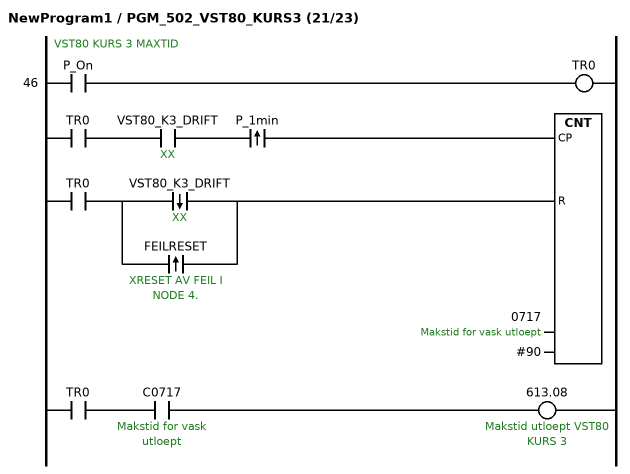
; [picture p552: NewProgram1 / PGM_502_VST80_KURS3, rungs 46-46]
; rung 46: VST80 KURS 3 MAXTID
LD P_On
OUT TR0
AND VST80_K3_DRIFT  ; XX
@AND P_1min
LD TR0
%LD VST80_K3_DRIFT  ; XX
@OR FEILRESET  ; XRESET AV FEIL I NODE 4.
ANDLD
CNT 0717 #90  ; Makstid for vask utloept
LD TR0
AND C0717  ; Makstid for vask utloept
OUT 613.08  ; Makstid utloept VST80 KURS 3

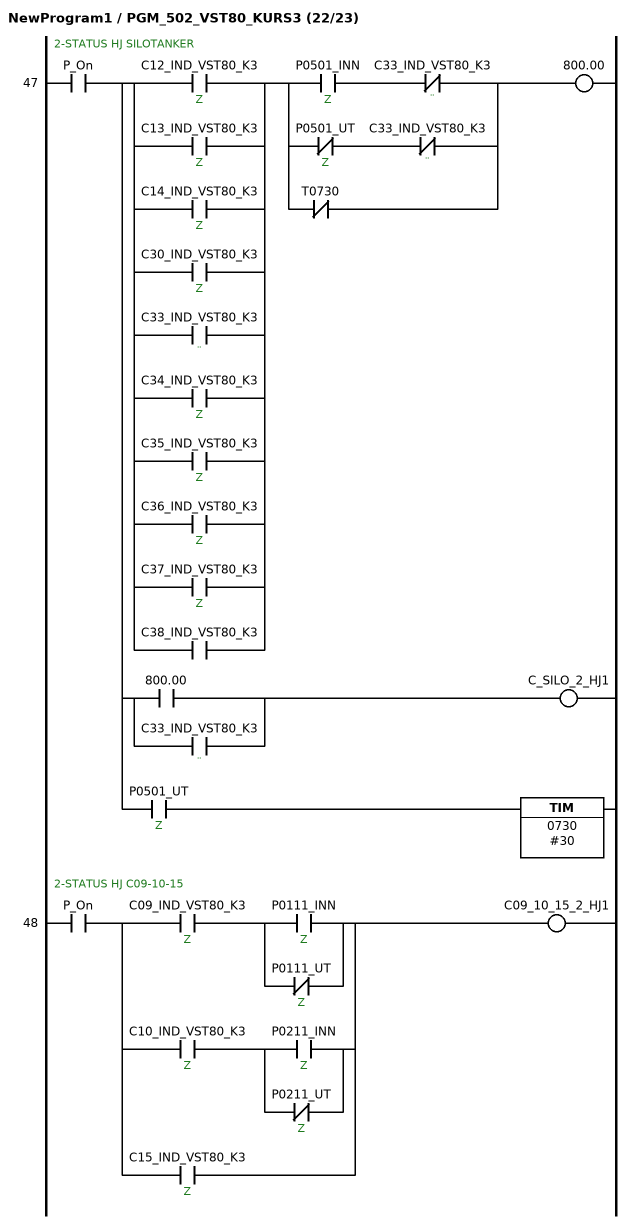
; rung 47: 2-STATUS HJ SILOTANKER
LD P_On
OUT TR0
LD C12_IND_VST80_K3  ; Z
OR C13_IND_VST80_K3  ; Z
OR C14_IND_VST80_K3  ; Z
OR C30_IND_VST80_K3  ; Z
OR C33_IND_VST80_K3  ; ¨
OR C34_IND_VST80_K3  ; Z
OR C35_IND_VST80_K3  ; Z
OR C36_IND_VST80_K3  ; Z
OR C37_IND_VST80_K3  ; Z
OR C38_IND_VST80_K3
ANDLD
LD P0501_INN  ; Z
ANDNOT C33_IND_VST80_K3  ; ¨
LDNOT P0501_UT  ; Z
ANDNOT C33_IND_VST80_K3  ; ¨
ORLD
ORNOT T0730
ANDLD
OUT 800.00
LD TR0
LD 800.00
OR C33_IND_VST80_K3  ; ¨
ANDLD
OUT C_SILO_2_HJ1
LD TR0
AND P0501_UT  ; Z
TIM 0730 #30
; rung 48: 2-STATUS HJ C09-10-15
LD P_On
LD C09_IND_VST80_K3  ; Z
LD P0111_INN  ; Z
ORNOT P0111_UT  ; Z
ANDLD
LD C10_IND_VST80_K3  ; Z
LD P0211_INN  ; Z
ORNOT P0211_UT  ; Z
ANDLD
ORLD
OR C15_IND_VST80_K3  ; Z
ANDLD
OUT C09_10_15_2_HJ1

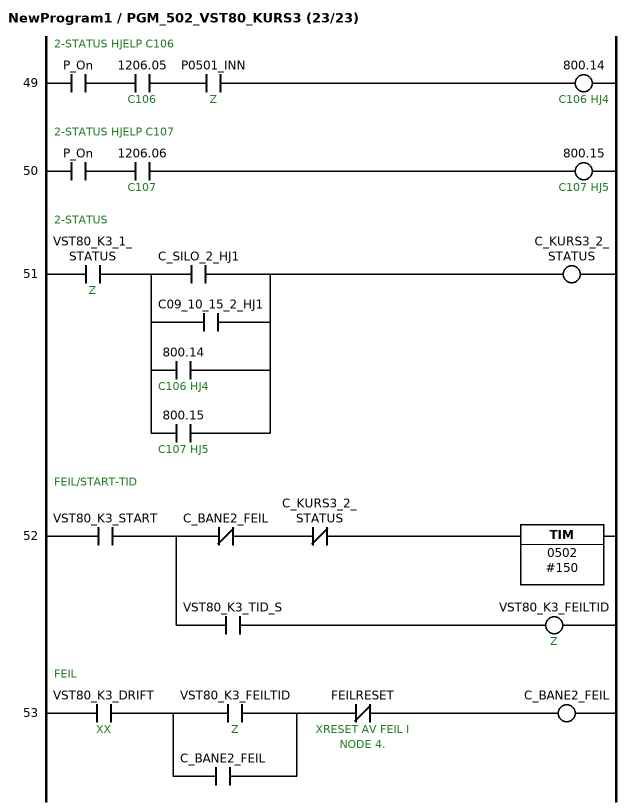
; rung 49: 2-STATUS HJELP C106
LD P_On
AND 1206.05  ; C106
AND P0501_INN  ; Z
OUT 800.14  ; C106 HJ4
; rung 50: 2-STATUS HJELP C107
LD P_On
AND 1206.06  ; C107
OUT 800.15  ; C107 HJ5
; rung 51: 2-STATUS
LD VST80_K3_1_STATUS  ; Z
LD C_SILO_2_HJ1
OR C09_10_15_2_HJ1
OR 800.14  ; C106 HJ4
OR 800.15  ; C107 HJ5
ANDLD
OUT C_KURS3_2_STATUS
; rung 52: FEIL/START-TID
LD VST80_K3_START
OUT TR0
ANDNOT C_BANE2_FEIL
ANDNOT C_KURS3_2_STATUS
TIM 0502 #150
LD TR0
AND VST80_K3_TID_S
OUT VST80_K3_FEILTID  ; Z
; rung 53: FEIL
LD VST80_K3_DRIFT  ; XX
LD VST80_K3_FEILTID  ; Z
OR C_BANE2_FEIL
ANDLD
ANDNOT FEILRESET  ; XRESET AV FEIL I NODE 4.
OUT C_BANE2_FEIL
; rung 54: Ingen_kommentar_funnet

### Section PGM503_C23

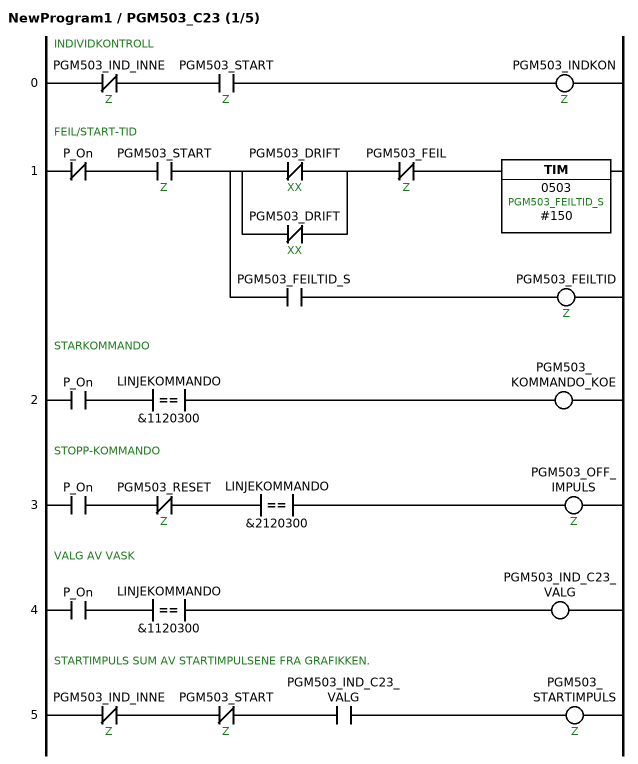
; rung 0: INDIVIDKONTROLL
LDNOT PGM503_IND_INNE  ; Z
AND PGM503_START  ; Z
OUT PGM503_INDKON  ; Z
; rung 1: FEIL/START-TID
LDNOT P_On
AND PGM503_START  ; Z
OUT TR0
LDNOT PGM503_DRIFT  ; XX
ORNOT PGM503_DRIFT  ; XX
ANDLD
ANDNOT PGM503_FEIL  ; Z
TIM 0503 #150  ; PGM503_FEILTID_S
LD TR0
AND PGM503_FEILTID_S
OUT PGM503_FEILTID  ; Z
; rung 2: STARKOMMANDO
LD P_On
AND=L(301) LINJEKOMMANDO &1120300
OUT PGM503_KOMMANDO_KOE
; rung 3: STOPP-KOMMANDO
LD P_On
ANDNOT PGM503_RESET  ; Z
AND=L(301) LINJEKOMMANDO &2120300
OUT PGM503_OFF_IMPULS  ; Z
; rung 4: VALG AV VASK
LD P_On
AND=L(301) LINJEKOMMANDO &1120300
OUT PGM503_IND_C23_VALG
; rung 5: STARTIMPULS SUM AV STARTIMPULSENE FRA GRAFIKKEN.
LDNOT PGM503_IND_INNE  ; Z
ANDNOT PGM503_START  ; Z
AND PGM503_IND_C23_VALG
OUT PGM503_STARTIMPULS  ; Z

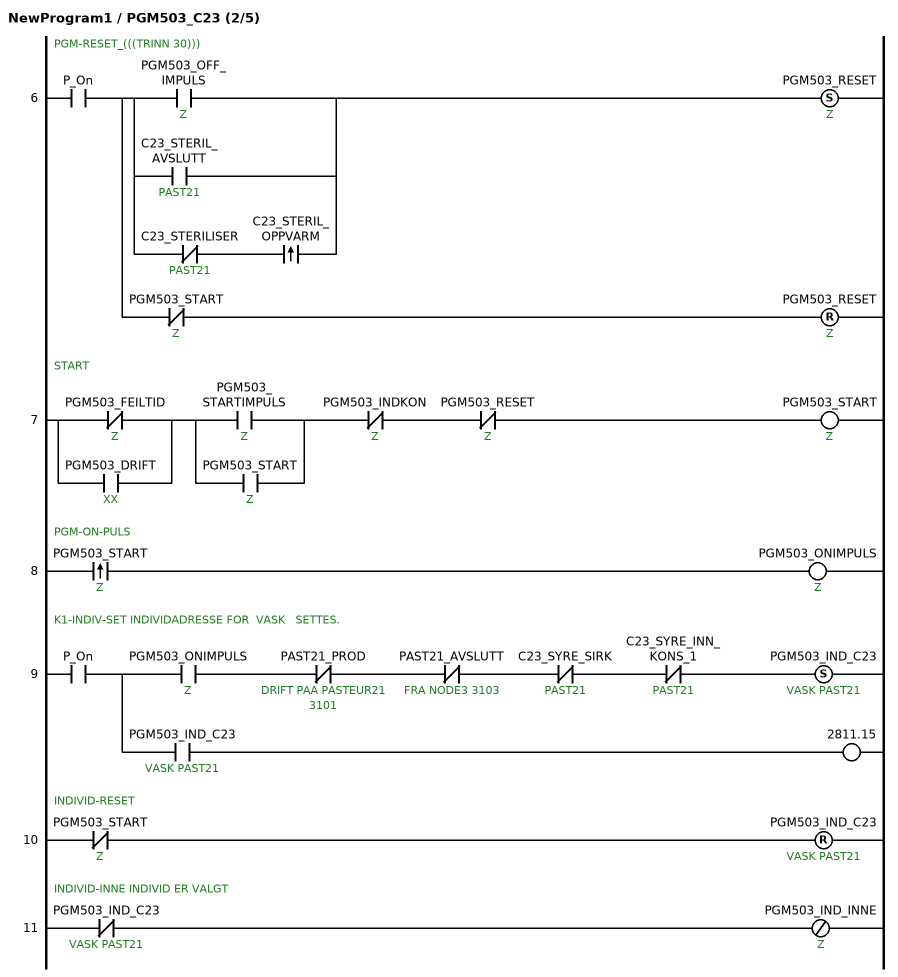
; rung 6: PGM-RESET_(((TRINN 30)))
LD P_On
OUT TR0
LD PGM503_OFF_IMPULS  ; Z
OR C23_STERIL_AVSLUTT  ; PAST21
LDNOT C23_STERILISER  ; PAST21
@AND C23_STERIL_OPPVARM
ORLD
ANDLD
SET PGM503_RESET  ; Z
LD TR0
ANDNOT PGM503_START  ; Z
RSET PGM503_RESET  ; Z
; rung 7: START
LDNOT PGM503_FEILTID  ; Z
OR PGM503_DRIFT  ; XX
LD PGM503_STARTIMPULS  ; Z
OR PGM503_START  ; Z
ANDLD
ANDNOT PGM503_INDKON  ; Z
ANDNOT PGM503_RESET  ; Z
OUT PGM503_START  ; Z
; rung 8: PGM-ON-PULS
@LD PGM503_START  ; Z
OUT PGM503_ONIMPULS  ; Z
; rung 9: K1-INDIV-SET INDIVIDADRESSE FOR  VASK   SETTES.
LD P_On
OUT TR0
AND PGM503_ONIMPULS  ; Z
ANDNOT PAST21_PROD  ; DRIFT PAA PASTEUR21 3101
ANDNOT PAST21_AVSLUTT  ; FRA NODE3 3103
ANDNOT C23_SYRE_SIRK  ; PAST21
ANDNOT C23_SYRE_INN_KONS_1  ; PAST21
SET PGM503_IND_C23  ; VASK PAST21
LD TR0
AND PGM503_IND_C23  ; VASK PAST21
OUT 2811.15
; rung 10: INDIVID-RESET
LDNOT PGM503_START  ; Z
RSET PGM503_IND_C23  ; VASK PAST21
; rung 11: INDIVID-INNE INDIVID ER VALGT
LDNOT PGM503_IND_C23  ; VASK PAST21
OUTNOT PGM503_IND_INNE  ; Z

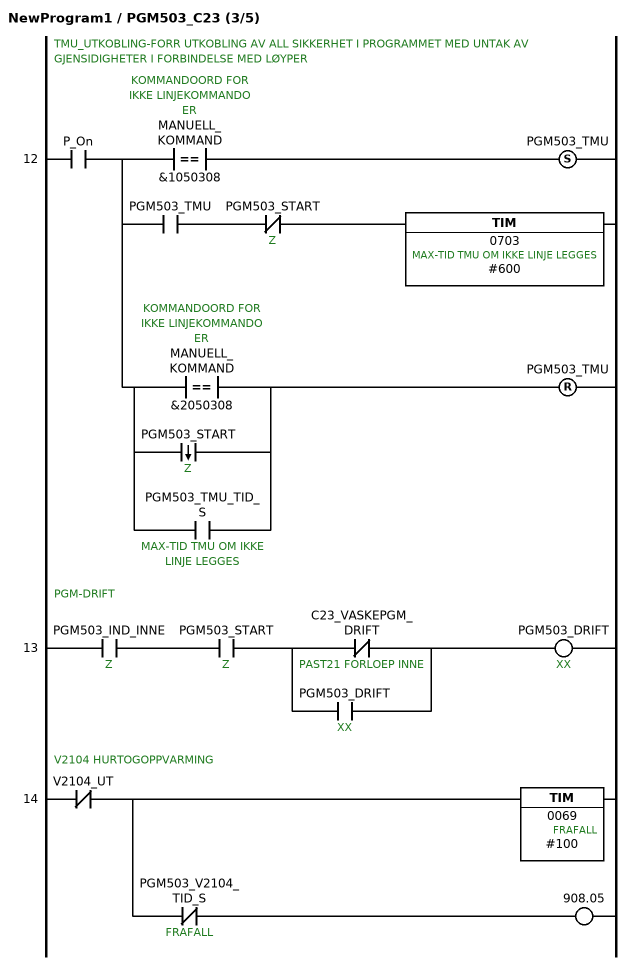
; rung 12: TMU_UTKOBLING-FORR UTKOBLING AV ALL SIKKERHET I PROGRAMMET MED UNTAK AV GJENSIDIGHETER I FORBINDELSE MED LØYPER
LD P_On
OUT TR0
AND=L(301) MANUELL_KOMMAND &1050308  ; KOMMANDOORD FOR IKKE LINJEKOMMANDOER
SET PGM503_TMU
LD TR0
AND PGM503_TMU
ANDNOT PGM503_START  ; Z
TIM 0703 #600  ; MAX-TID TMU OM IKKE LINJE LEGGES
LD TR0
LD=L(301) MANUELL_KOMMAND &2050308  ; KOMMANDOORD FOR IKKE LINJEKOMMANDOER
%OR PGM503_START  ; Z
OR PGM503_TMU_TID_S  ; MAX-TID TMU OM IKKE LINJE LEGGES
ANDLD
RSET PGM503_TMU
; rung 13: PGM-DRIFT
LD PGM503_IND_INNE  ; Z
AND PGM503_START  ; Z
LDNOT C23_VASKEPGM_DRIFT  ; PAST21 FORLOEP INNE
OR PGM503_DRIFT  ; XX
ANDLD
OUT PGM503_DRIFT  ; XX
; rung 14: V2104 HURTOGOPPVARMING
LDNOT V2104_UT
TIM 0069 #100  ; FRAFALL
ANDNOT PGM503_V2104_TID_S  ; FRAFALL
OUT 908.05

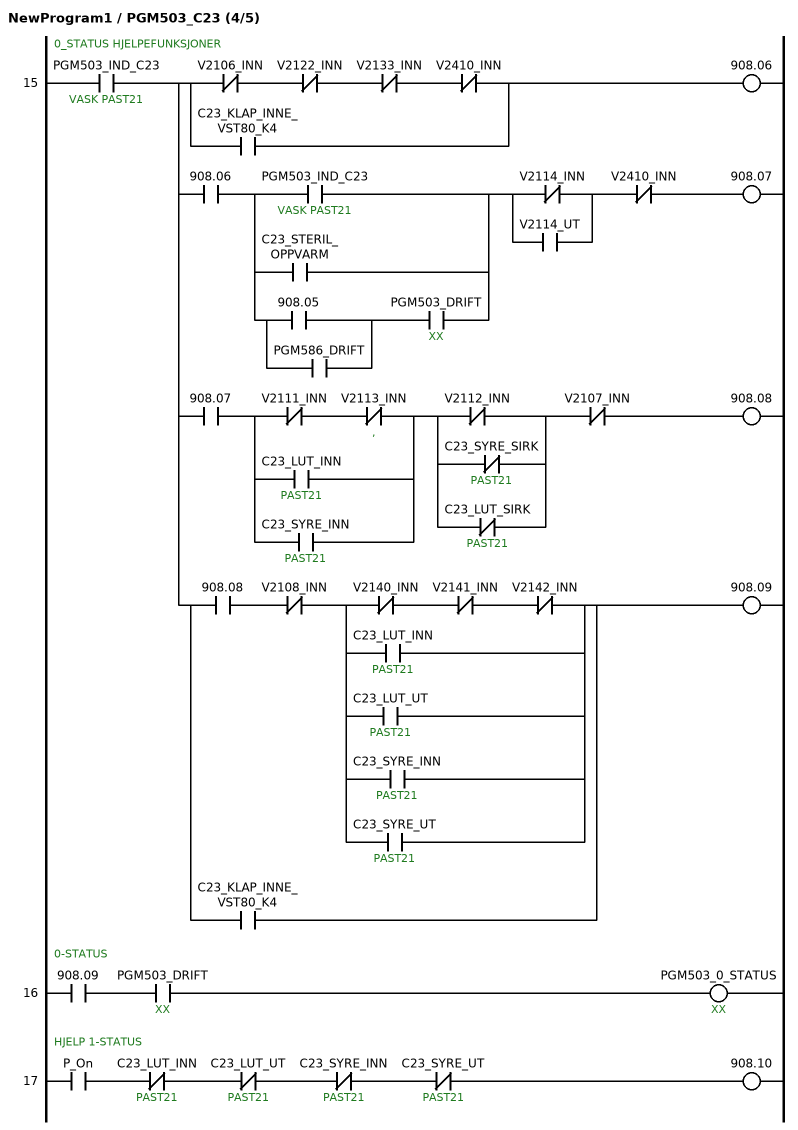
; rung 15: 0_STATUS HJELPEFUNKSJONER
LD PGM503_IND_C23  ; VASK PAST21
OUT TR0
LDNOT V2106_INN
ANDNOT V2122_INN
ANDNOT V2133_INN
ANDNOT V2410_INN
OR C23_KLAP_INNE_VST80_K4
ANDLD
OUT 908.06
LD TR0
AND 908.06
LD PGM503_IND_C23  ; VASK PAST21
OR C23_STERIL_OPPVARM
LD 908.05
OR PGM586_DRIFT
AND PGM503_DRIFT  ; XX
ORLD
ANDLD
LDNOT V2114_INN
OR V2114_UT
ANDLD
ANDNOT V2410_INN
OUT 908.07
LD TR0
AND 908.07
LDNOT V2111_INN
ANDNOT V2113_INN  ; ,
OR C23_LUT_INN  ; PAST21
OR C23_SYRE_INN  ; PAST21
ANDLD
LDNOT V2112_INN
ORNOT C23_SYRE_SIRK  ; PAST21
ORNOT C23_LUT_SIRK  ; PAST21
ANDLD
ANDNOT V2107_INN
OUT 908.08
LD TR0
LD 908.08
ANDNOT V2108_INN
LDNOT V2140_INN
ANDNOT V2141_INN
ANDNOT V2142_INN
OR C23_LUT_INN  ; PAST21
OR C23_LUT_UT  ; PAST21
OR C23_SYRE_INN  ; PAST21
OR C23_SYRE_UT  ; PAST21
ANDLD
OR C23_KLAP_INNE_VST80_K4
ANDLD
OUT 908.09
; rung 16: 0-STATUS
LD 908.09
AND PGM503_DRIFT  ; XX
OUT PGM503_0_STATUS  ; XX
; rung 17: HJELP 1-STATUS
LD P_On
ANDNOT C23_LUT_INN  ; PAST21
ANDNOT C23_LUT_UT  ; PAST21
ANDNOT C23_SYRE_INN  ; PAST21
ANDNOT C23_SYRE_UT  ; PAST21
OUT 908.10

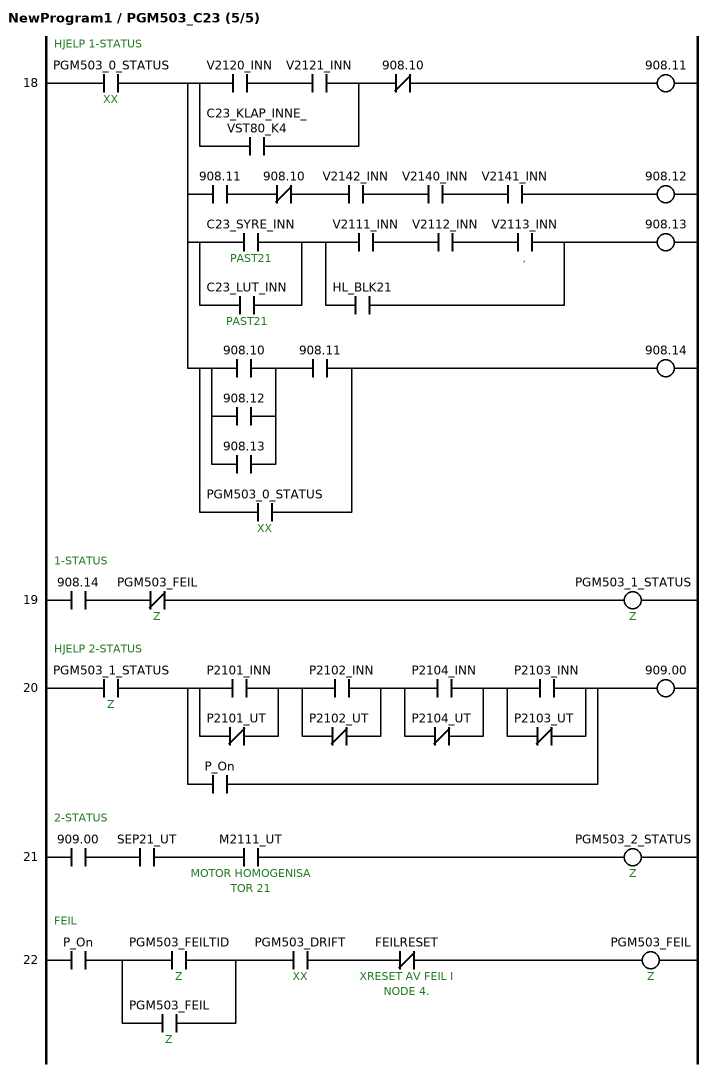
; rung 18: HJELP 1-STATUS
LD PGM503_0_STATUS  ; XX
OUT TR0
LD V2120_INN
AND V2121_INN
OR C23_KLAP_INNE_VST80_K4
ANDLD
ANDNOT 908.10
OUT 908.11
LD TR0
AND 908.11
ANDNOT 908.10
AND V2142_INN
AND V2140_INN
AND V2141_INN
OUT 908.12
LD TR0
LD C23_SYRE_INN  ; PAST21
OR C23_LUT_INN  ; PAST21
ANDLD
LD V2111_INN
AND V2112_INN
AND V2113_INN  ; ,
OR HL_BLK21
ANDLD
OUT 908.13
LD TR0
LD 908.10
OR 908.12
OR 908.13
AND 908.11
OR PGM503_0_STATUS  ; XX
ANDLD
OUT 908.14
; rung 19: 1-STATUS
LD 908.14
ANDNOT PGM503_FEIL  ; Z
OUT PGM503_1_STATUS  ; Z
; rung 20: HJELP 2-STATUS
LD PGM503_1_STATUS  ; Z
LD P2101_INN
ORNOT P2101_UT
LD P2102_INN
ORNOT P2102_UT
ANDLD
LD P2104_INN
ORNOT P2104_UT
ANDLD
LD P2103_INN
ORNOT P2103_UT
ANDLD
OR P_On
ANDLD
OUT 909.00
; rung 21: 2-STATUS
LD 909.00
AND SEP21_UT
AND M2111_UT  ; MOTOR HOMOGENISATOR 21
OUT PGM503_2_STATUS  ; Z
; rung 22: FEIL
LD P_On
LD PGM503_FEILTID  ; Z
OR PGM503_FEIL  ; Z
ANDLD
AND PGM503_DRIFT  ; XX
ANDNOT FEILRESET  ; XRESET AV FEIL I NODE 4.
OUT PGM503_FEIL  ; Z
; rung 23: Ingen_kommentar_funnet

### Section C23_KLAPRING

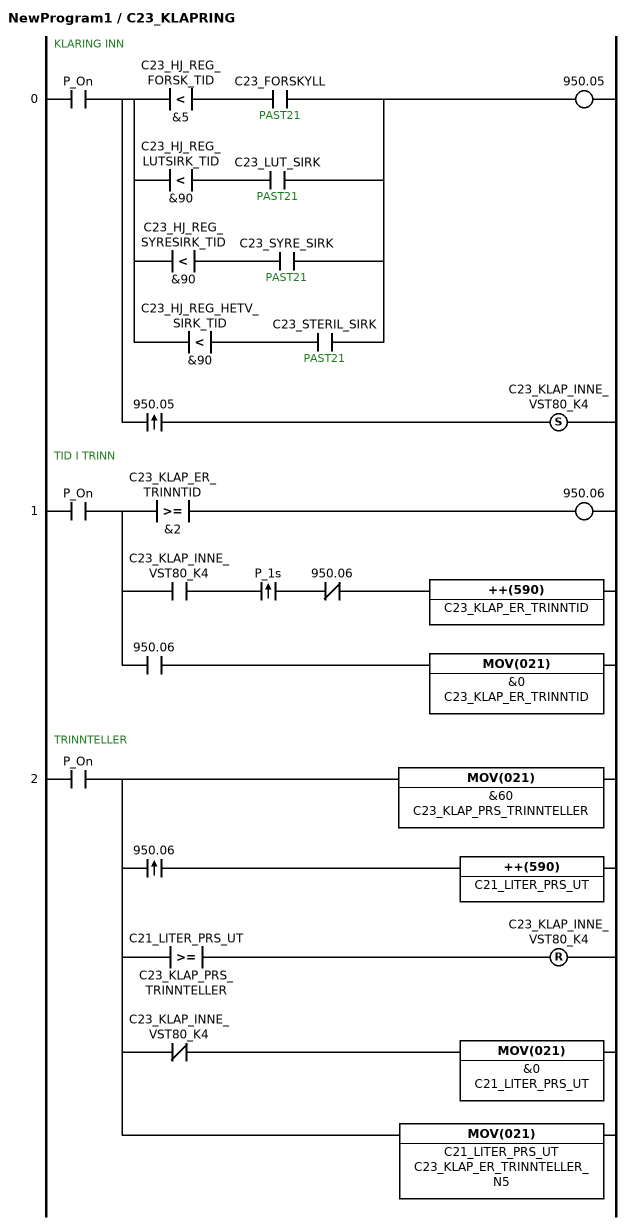
; rung 0: KLARING INN
LD P_On
OUT TR0
LD<(310) C23_HJ_REG_FORSK_TID &5
AND C23_FORSKYLL  ; PAST21
LD<(310) C23_HJ_REG_LUTSIRK_TID &90
AND C23_LUT_SIRK  ; PAST21
ORLD
LD<(310) C23_HJ_REG_SYRESIRK_TID &90
AND C23_SYRE_SIRK  ; PAST21
ORLD
LD<(310) C23_HJ_REG_HETV_SIRK_TID &90
AND C23_STERIL_SIRK  ; PAST21
ORLD
ANDLD
OUT 950.05
LD TR0
@AND 950.05
SET C23_KLAP_INNE_VST80_K4
; rung 1: TID I TRINN
LD P_On
OUT TR0
AND>=(325) C23_KLAP_ER_TRINNTID &2
OUT 950.06
LD TR0
AND C23_KLAP_INNE_VST80_K4
@AND P_1s
ANDNOT 950.06
++(590) C23_KLAP_ER_TRINNTID
LD TR0
AND 950.06
MOV(021) &0 C23_KLAP_ER_TRINNTID
; rung 2: TRINNTELLER
LD P_On
OUT TR0
MOV(021) &60 C23_KLAP_PRS_TRINNTELLER
@AND 950.06
++(590) C21_LITER_PRS_UT
LD TR0
AND>=(325) C21_LITER_PRS_UT C23_KLAP_PRS_TRINNTELLER
RSET C23_KLAP_INNE_VST80_K4
LD TR0
ANDNOT C23_KLAP_INNE_VST80_K4
MOV(021) &0 C21_LITER_PRS_UT
LD TR0
MOV(021) C21_LITER_PRS_UT C23_KLAP_ER_TRINNTELLER_N5
; rung 3: Ingen_kommentar_funnet

### Section PGM504_C24

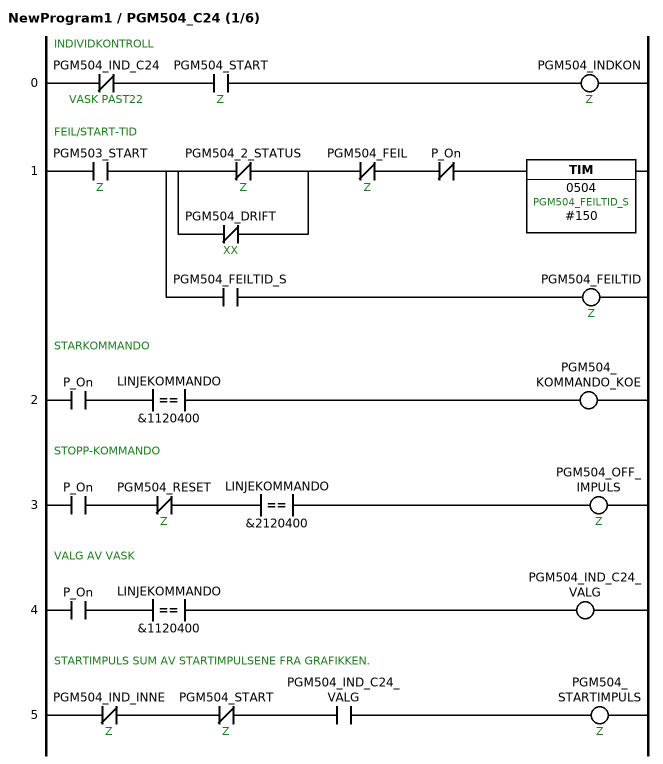
; rung 0: INDIVIDKONTROLL
LDNOT PGM504_IND_C24  ; VASK PAST22
AND PGM504_START  ; Z
OUT PGM504_INDKON  ; Z
; rung 1: FEIL/START-TID
LD PGM503_START  ; Z
OUT TR0
LDNOT PGM504_2_STATUS  ; Z
ORNOT PGM504_DRIFT  ; XX
ANDLD
ANDNOT PGM504_FEIL  ; Z
ANDNOT P_On
TIM 0504 #150  ; PGM504_FEILTID_S
LD TR0
AND PGM504_FEILTID_S
OUT PGM504_FEILTID  ; Z
; rung 2: STARKOMMANDO
LD P_On
AND=L(301) LINJEKOMMANDO &1120400
OUT PGM504_KOMMANDO_KOE
; rung 3: STOPP-KOMMANDO
LD P_On
ANDNOT PGM504_RESET  ; Z
AND=L(301) LINJEKOMMANDO &2120400
OUT PGM504_OFF_IMPULS  ; Z
; rung 4: VALG AV VASK
LD P_On
AND=L(301) LINJEKOMMANDO &1120400
OUT PGM504_IND_C24_VALG
; rung 5: STARTIMPULS SUM AV STARTIMPULSENE FRA GRAFIKKEN.
LDNOT PGM504_IND_INNE  ; Z
ANDNOT PGM504_START  ; Z
AND PGM504_IND_C24_VALG
OUT PGM504_STARTIMPULS  ; Z

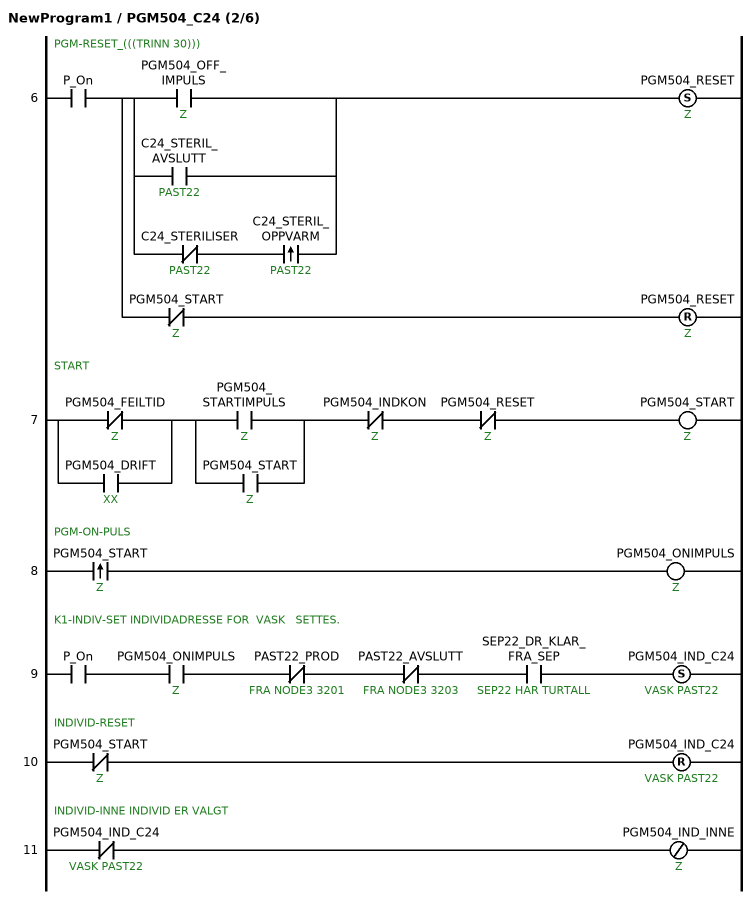
; rung 6: PGM-RESET_(((TRINN 30)))
LD P_On
OUT TR0
LD PGM504_OFF_IMPULS  ; Z
OR C24_STERIL_AVSLUTT  ; PAST22
LDNOT C24_STERILISER  ; PAST22
@AND C24_STERIL_OPPVARM  ; PAST22
ORLD
ANDLD
SET PGM504_RESET  ; Z
LD TR0
ANDNOT PGM504_START  ; Z
RSET PGM504_RESET  ; Z
; rung 7: START
LDNOT PGM504_FEILTID  ; Z
OR PGM504_DRIFT  ; XX
LD PGM504_STARTIMPULS  ; Z
OR PGM504_START  ; Z
ANDLD
ANDNOT PGM504_INDKON  ; Z
ANDNOT PGM504_RESET  ; Z
OUT PGM504_START  ; Z
; rung 8: PGM-ON-PULS
@LD PGM504_START  ; Z
OUT PGM504_ONIMPULS  ; Z
; rung 9: K1-INDIV-SET INDIVIDADRESSE FOR  VASK   SETTES.
LD P_On
AND PGM504_ONIMPULS  ; Z
ANDNOT PAST22_PROD  ; FRA NODE3 3201
ANDNOT PAST22_AVSLUTT  ; FRA NODE3 3203
AND SEP22_DR_KLAR_FRA_SEP  ; SEP22 HAR TURTALL
SET PGM504_IND_C24  ; VASK PAST22
; rung 10: INDIVID-RESET
LDNOT PGM504_START  ; Z
RSET PGM504_IND_C24  ; VASK PAST22
; rung 11: INDIVID-INNE INDIVID ER VALGT
LDNOT PGM504_IND_C24  ; VASK PAST22
OUTNOT PGM504_IND_INNE  ; Z

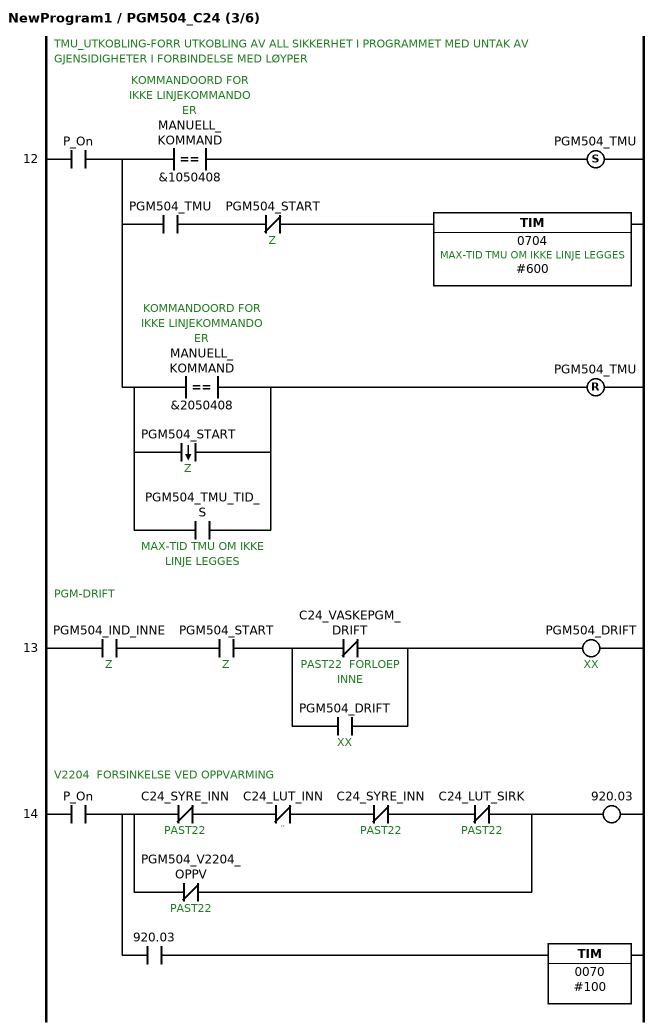
; rung 12: TMU_UTKOBLING-FORR UTKOBLING AV ALL SIKKERHET I PROGRAMMET MED UNTAK AV GJENSIDIGHETER I FORBINDELSE MED LØYPER
LD P_On
OUT TR0
AND=L(301) MANUELL_KOMMAND &1050408  ; KOMMANDOORD FOR IKKE LINJEKOMMANDOER
SET PGM504_TMU
LD TR0
AND PGM504_TMU
ANDNOT PGM504_START  ; Z
TIM 0704 #600  ; MAX-TID TMU OM IKKE LINJE LEGGES
LD TR0
LD=L(301) MANUELL_KOMMAND &2050408  ; KOMMANDOORD FOR IKKE LINJEKOMMANDOER
%OR PGM504_START  ; Z
OR PGM504_TMU_TID_S  ; MAX-TID TMU OM IKKE LINJE LEGGES
ANDLD
RSET PGM504_TMU
; rung 13: PGM-DRIFT
LD PGM504_IND_INNE  ; Z
AND PGM504_START  ; Z
LDNOT C24_VASKEPGM_DRIFT  ; PAST22  FORLOEP INNE
OR PGM504_DRIFT  ; XX
ANDLD
OUT PGM504_DRIFT  ; XX
; rung 14: V2204  FORSINKELSE VED OPPVARMING
LD P_On
OUT TR0
LDNOT C24_SYRE_INN  ; PAST22
ANDNOT C24_LUT_INN  ; ¨
ANDNOT C24_SYRE_INN  ; PAST22
ANDNOT C24_LUT_SIRK  ; PAST22
ORNOT PGM504_V2204_OPPV  ; PAST22
ANDLD
OUT 920.03
LD TR0
AND 920.03
TIM 0070 #100

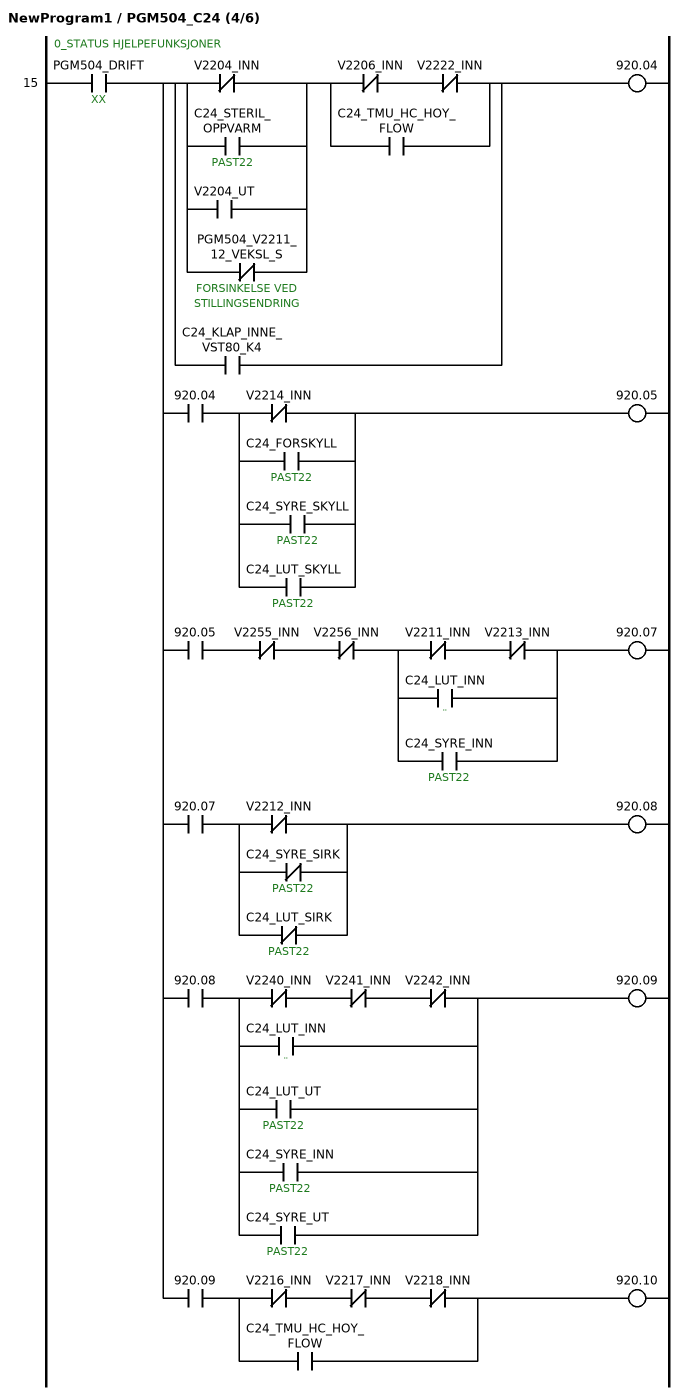
; rung 15: 0_STATUS HJELPEFUNKSJONER
LD PGM504_DRIFT  ; XX
OUT TR0
LDNOT V2204_INN
OR C24_STERIL_OPPVARM  ; PAST22
OR V2204_UT
ORNOT PGM504_V2211_12_VEKSL_S  ; FORSINKELSE VED STILLINGSENDRING
LDNOT V2206_INN
ANDNOT V2222_INN
OR C24_TMU_HC_HOY_FLOW
ANDLD
OR C24_KLAP_INNE_VST80_K4
ANDLD
OUT 920.04
LD TR0
AND 920.04
LDNOT V2214_INN
OR C24_FORSKYLL  ; PAST22
OR C24_SYRE_SKYLL  ; PAST22
OR C24_LUT_SKYLL  ; PAST22
ANDLD
OUT 920.05
LD TR0
AND 920.05
ANDNOT V2255_INN
ANDNOT V2256_INN
LDNOT V2211_INN
ANDNOT V2213_INN
OR C24_LUT_INN  ; ¨
OR C24_SYRE_INN  ; PAST22
ANDLD
OUT 920.07
LD TR0
AND 920.07
LDNOT V2212_INN
ORNOT C24_SYRE_SIRK  ; PAST22
ORNOT C24_LUT_SIRK  ; PAST22
ANDLD
OUT 920.08
LD TR0
AND 920.08
LDNOT V2240_INN
ANDNOT V2241_INN
ANDNOT V2242_INN
OR C24_LUT_INN  ; ¨
OR C24_LUT_UT  ; PAST22
OR C24_SYRE_INN  ; PAST22
OR C24_SYRE_UT  ; PAST22
ANDLD
OUT 920.09
LD TR0
AND 920.09
LDNOT V2216_INN
ANDNOT V2217_INN
ANDNOT V2218_INN
OR C24_TMU_HC_HOY_FLOW
ANDLD
OUT 920.10

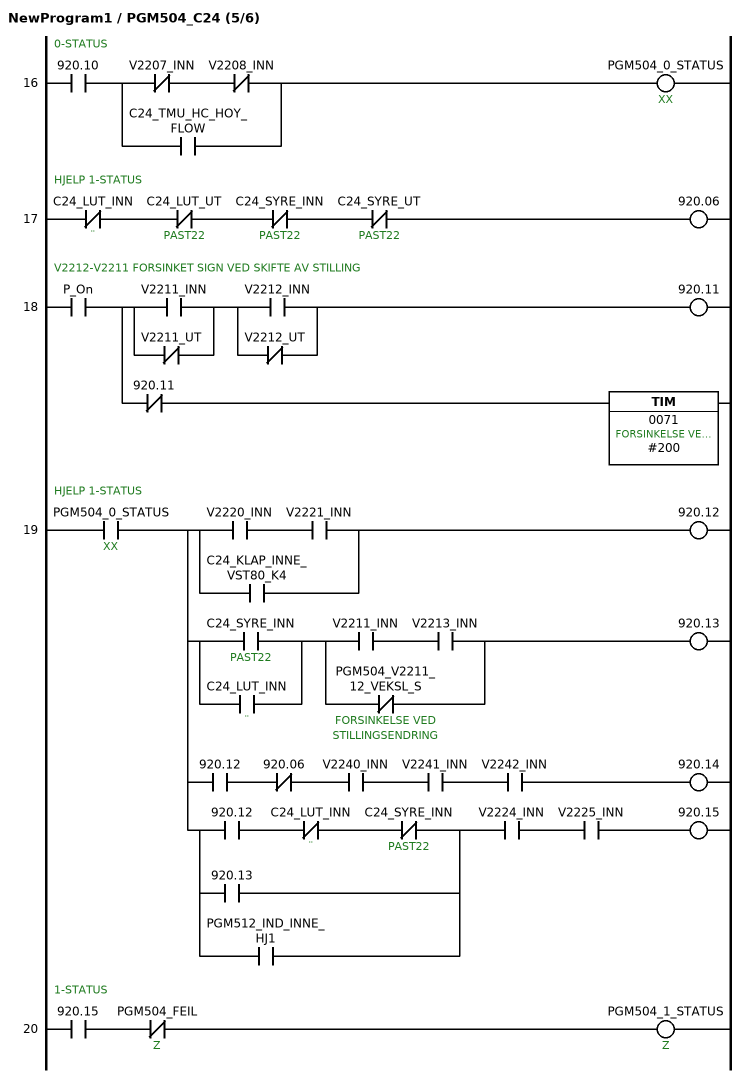
; rung 16: 0-STATUS
LD 920.10
LDNOT V2207_INN
ANDNOT V2208_INN
OR C24_TMU_HC_HOY_FLOW
ANDLD
OUT PGM504_0_STATUS  ; XX
; rung 17: HJELP 1-STATUS
LDNOT C24_LUT_INN  ; ¨
ANDNOT C24_LUT_UT  ; PAST22
ANDNOT C24_SYRE_INN  ; PAST22
ANDNOT C24_SYRE_UT  ; PAST22
OUT 920.06
; rung 18: V2212-V2211 FORSINKET SIGN VED SKIFTE AV STILLING
LD P_On
OUT TR0
LD V2211_INN
ORNOT V2211_UT
ANDLD
LD V2212_INN
ORNOT V2212_UT
ANDLD
OUT 920.11
LD TR0
ANDNOT 920.11
TIM 0071 #200  ; FORSINKELSE VED STILLINGSENDRING
; rung 19: HJELP 1-STATUS
LD PGM504_0_STATUS  ; XX
OUT TR0
LD V2220_INN
AND V2221_INN
OR C24_KLAP_INNE_VST80_K4
ANDLD
OUT 920.12
LD TR0
LD C24_SYRE_INN  ; PAST22
OR C24_LUT_INN  ; ¨
ANDLD
LD V2211_INN
AND V2213_INN
ORNOT PGM504_V2211_12_VEKSL_S  ; FORSINKELSE VED STILLINGSENDRING
ANDLD
OUT 920.13
LD TR0
AND 920.12
ANDNOT 920.06
AND V2240_INN
AND V2241_INN
AND V2242_INN
OUT 920.14
LD TR0
LD 920.12
ANDNOT C24_LUT_INN  ; ¨
ANDNOT C24_SYRE_INN  ; PAST22
OR 920.13
OR PGM512_IND_INNE_HJ1
ANDLD
AND V2224_INN
AND V2225_INN
OUT 920.15
; rung 20: 1-STATUS
LD 920.15
ANDNOT PGM504_FEIL  ; Z
OUT PGM504_1_STATUS  ; Z

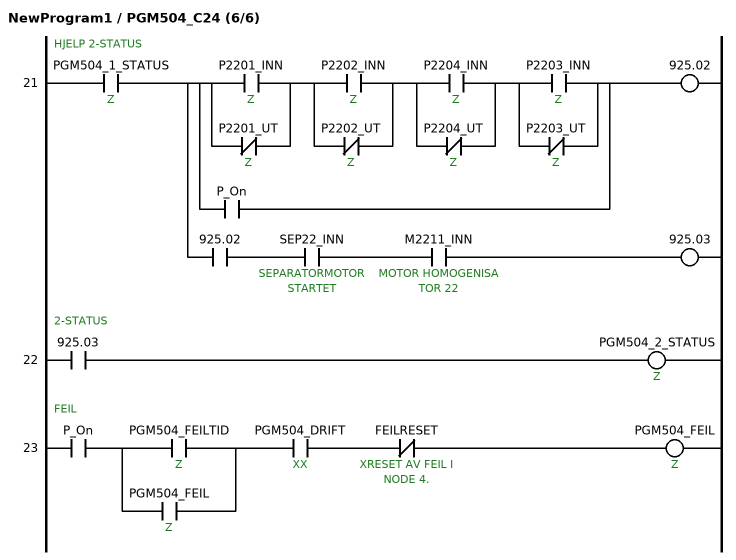
; rung 21: HJELP 2-STATUS
LD PGM504_1_STATUS  ; Z
OUT TR0
LD P2201_INN  ; Z
ORNOT P2201_UT  ; Z
LD P2202_INN  ; Z
ORNOT P2202_UT  ; Z
ANDLD
LD P2204_INN  ; Z
ORNOT P2204_UT  ; Z
ANDLD
LD P2203_INN  ; Z
ORNOT P2203_UT  ; Z
ANDLD
OR P_On
ANDLD
OUT 925.02
LD TR0
AND 925.02
AND SEP22_INN  ; SEPARATORMOTOR STARTET
AND M2211_INN  ; MOTOR HOMOGENISATOR 22
OUT 925.03
; rung 22: 2-STATUS
LD 925.03
OUT PGM504_2_STATUS  ; Z
; rung 23: FEIL
LD P_On
LD PGM504_FEILTID  ; Z
OR PGM504_FEIL  ; Z
ANDLD
AND PGM504_DRIFT  ; XX
ANDNOT FEILRESET  ; XRESET AV FEIL I NODE 4.
OUT PGM504_FEIL  ; Z
; rung 24: Ingen_kommentar_funnet

### Section C24_KLAPRING

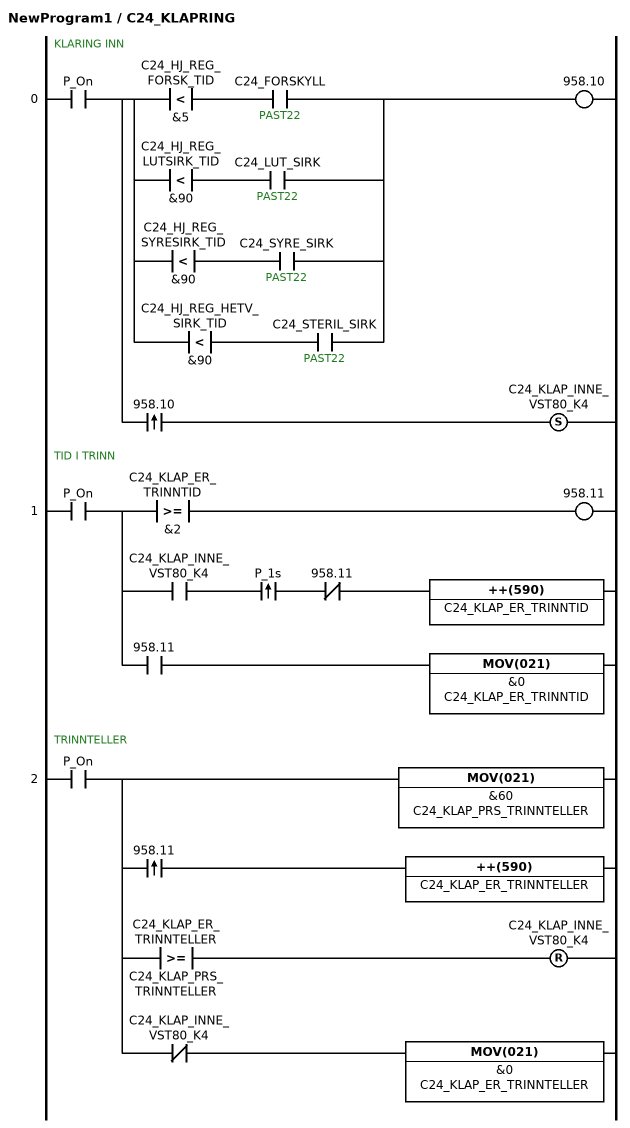
; rung 0: KLARING INN
LD P_On
OUT TR0
LD<(310) C24_HJ_REG_FORSK_TID &5
AND C24_FORSKYLL  ; PAST22
LD<(310) C24_HJ_REG_LUTSIRK_TID &90
AND C24_LUT_SIRK  ; PAST22
ORLD
LD<(310) C24_HJ_REG_SYRESIRK_TID &90
AND C24_SYRE_SIRK  ; PAST22
ORLD
LD<(310) C24_HJ_REG_HETV_SIRK_TID &90
AND C24_STERIL_SIRK  ; PAST22
ORLD
ANDLD
OUT 958.10
LD TR0
@AND 958.10
SET C24_KLAP_INNE_VST80_K4
; rung 1: TID I TRINN
LD P_On
OUT TR0
AND>=(325) C24_KLAP_ER_TRINNTID &2
OUT 958.11
LD TR0
AND C24_KLAP_INNE_VST80_K4
@AND P_1s
ANDNOT 958.11
++(590) C24_KLAP_ER_TRINNTID
LD TR0
AND 958.11
MOV(021) &0 C24_KLAP_ER_TRINNTID
; rung 2: TRINNTELLER
LD P_On
OUT TR0
MOV(021) &60 C24_KLAP_PRS_TRINNTELLER
@AND 958.11
++(590) C24_KLAP_ER_TRINNTELLER
LD TR0
AND>=(325) C24_KLAP_ER_TRINNTELLER C24_KLAP_PRS_TRINNTELLER
RSET C24_KLAP_INNE_VST80_K4
LD TR0
ANDNOT C24_KLAP_INNE_VST80_K4
MOV(021) &0 C24_KLAP_ER_TRINNTELLER
; rung 3: Ingen_kommentar_funnet

### Section PGM505_C25

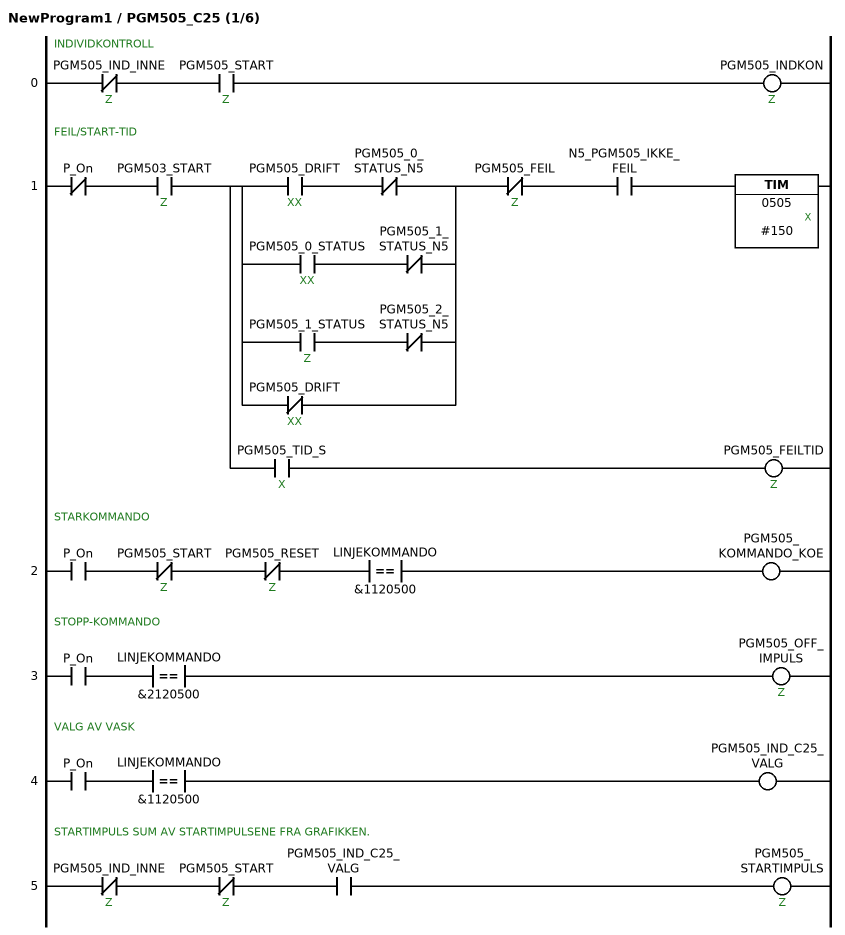
; rung 0: INDIVIDKONTROLL
LDNOT PGM505_IND_INNE  ; Z
AND PGM505_START  ; Z
OUT PGM505_INDKON  ; Z
; rung 1: FEIL/START-TID
LDNOT P_On
AND PGM503_START  ; Z
OUT TR0
LD PGM505_DRIFT  ; XX
ANDNOT PGM505_0_STATUS_N5
LD PGM505_0_STATUS  ; XX
ANDNOT PGM505_1_STATUS_N5
ORLD
LD PGM505_1_STATUS  ; Z
ANDNOT PGM505_2_STATUS_N5
ORLD
ORNOT PGM505_DRIFT  ; XX
ANDLD
ANDNOT PGM505_FEIL  ; Z
AND N5_PGM505_IKKE_FEIL
TIM 0505 #150  ; X
LD TR0
AND PGM505_TID_S  ; X
OUT PGM505_FEILTID  ; Z
; rung 2: STARKOMMANDO
LD P_On
ANDNOT PGM505_START  ; Z
ANDNOT PGM505_RESET  ; Z
AND=L(301) LINJEKOMMANDO &1120500
OUT PGM505_KOMMANDO_KOE
; rung 3: STOPP-KOMMANDO
LD P_On
AND=L(301) LINJEKOMMANDO &2120500
OUT PGM505_OFF_IMPULS  ; Z
; rung 4: VALG AV VASK
LD P_On
AND=L(301) LINJEKOMMANDO &1120500
OUT PGM505_IND_C25_VALG
; rung 5: STARTIMPULS SUM AV STARTIMPULSENE FRA GRAFIKKEN.
LDNOT PGM505_IND_INNE  ; Z
ANDNOT PGM505_START  ; Z
AND PGM505_IND_C25_VALG
OUT PGM505_STARTIMPULS  ; Z

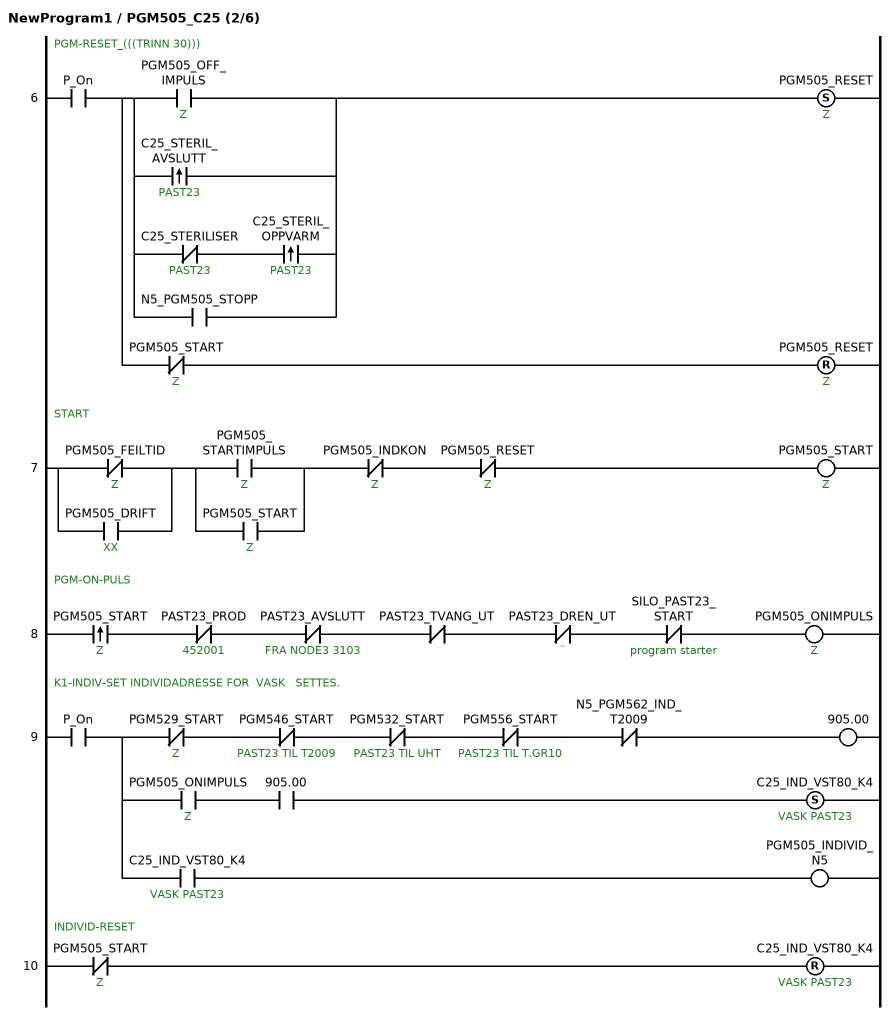
; rung 6: PGM-RESET_(((TRINN 30)))
LD P_On
OUT TR0
LD PGM505_OFF_IMPULS  ; Z
@OR C25_STERIL_AVSLUTT  ; PAST23
LDNOT C25_STERILISER  ; PAST23
@AND C25_STERIL_OPPVARM  ; PAST23
ORLD
OR N5_PGM505_STOPP
ANDLD
SET PGM505_RESET  ; Z
LD TR0
ANDNOT PGM505_START  ; Z
RSET PGM505_RESET  ; Z
; rung 7: START
LDNOT PGM505_FEILTID  ; Z
OR PGM505_DRIFT  ; XX
LD PGM505_STARTIMPULS  ; Z
OR PGM505_START  ; Z
ANDLD
ANDNOT PGM505_INDKON  ; Z
ANDNOT PGM505_RESET  ; Z
OUT PGM505_START  ; Z
; rung 8: PGM-ON-PULS
@LD PGM505_START  ; Z
ANDNOT PAST23_PROD  ; 452001
ANDNOT PAST23_AVSLUTT  ; FRA NODE3 3103
ANDNOT PAST23_TVANG_UT
ANDNOT PAST23_DREN_UT  ; ¨
ANDNOT SILO_PAST23_START  ; program starter
OUT PGM505_ONIMPULS  ; Z
; rung 9: K1-INDIV-SET INDIVIDADRESSE FOR  VASK   SETTES.
LD P_On
OUT TR0
ANDNOT PGM529_START  ; Z
ANDNOT PGM546_START  ; PAST23 TIL T2009
ANDNOT PGM532_START  ; PAST23 TIL UHT
ANDNOT PGM556_START  ; PAST23 TIL T.GR10
ANDNOT N5_PGM562_IND_T2009
OUT 905.00
LD TR0
AND PGM505_ONIMPULS  ; Z
AND 905.00
SET C25_IND_VST80_K4  ; VASK PAST23
LD TR0
AND C25_IND_VST80_K4  ; VASK PAST23
OUT PGM505_INDIVID_N5
; rung 10: INDIVID-RESET
LDNOT PGM505_START  ; Z
RSET C25_IND_VST80_K4  ; VASK PAST23

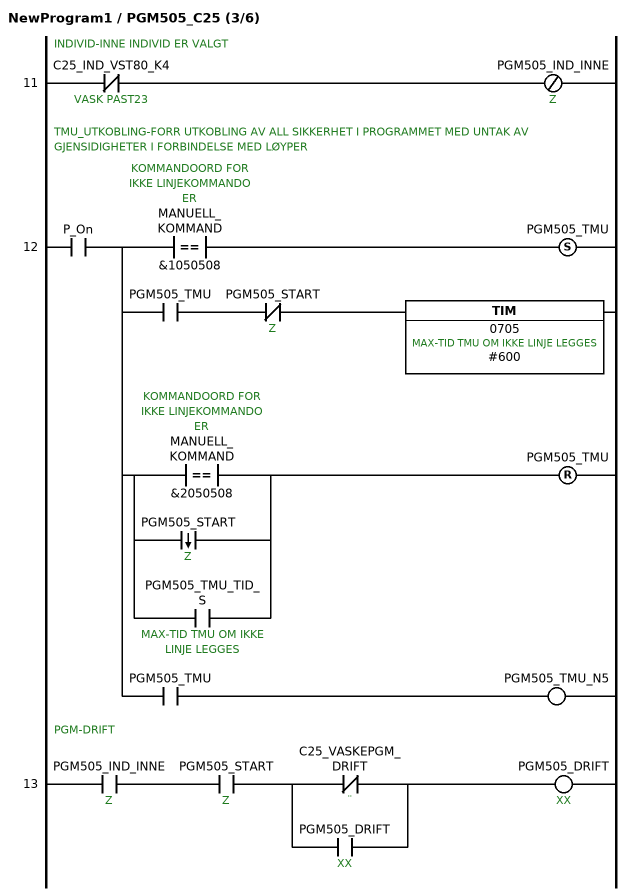
; rung 11: INDIVID-INNE INDIVID ER VALGT
LDNOT C25_IND_VST80_K4  ; VASK PAST23
OUTNOT PGM505_IND_INNE  ; Z
; rung 12: TMU_UTKOBLING-FORR UTKOBLING AV ALL SIKKERHET I PROGRAMMET MED UNTAK AV GJENSIDIGHETER I FORBINDELSE MED LØYPER
LD P_On
OUT TR0
AND=L(301) MANUELL_KOMMAND &1050508  ; KOMMANDOORD FOR IKKE LINJEKOMMANDOER
SET PGM505_TMU
LD TR0
AND PGM505_TMU
ANDNOT PGM505_START  ; Z
TIM 0705 #600  ; MAX-TID TMU OM IKKE LINJE LEGGES
LD TR0
LD=L(301) MANUELL_KOMMAND &2050508  ; KOMMANDOORD FOR IKKE LINJEKOMMANDOER
%OR PGM505_START  ; Z
OR PGM505_TMU_TID_S  ; MAX-TID TMU OM IKKE LINJE LEGGES
ANDLD
RSET PGM505_TMU
LD TR0
AND PGM505_TMU
OUT PGM505_TMU_N5
; rung 13: PGM-DRIFT
LD PGM505_IND_INNE  ; Z
AND PGM505_START  ; Z
LDNOT C25_VASKEPGM_DRIFT  ; ¨
OR PGM505_DRIFT  ; XX
ANDLD
OUT PGM505_DRIFT  ; XX

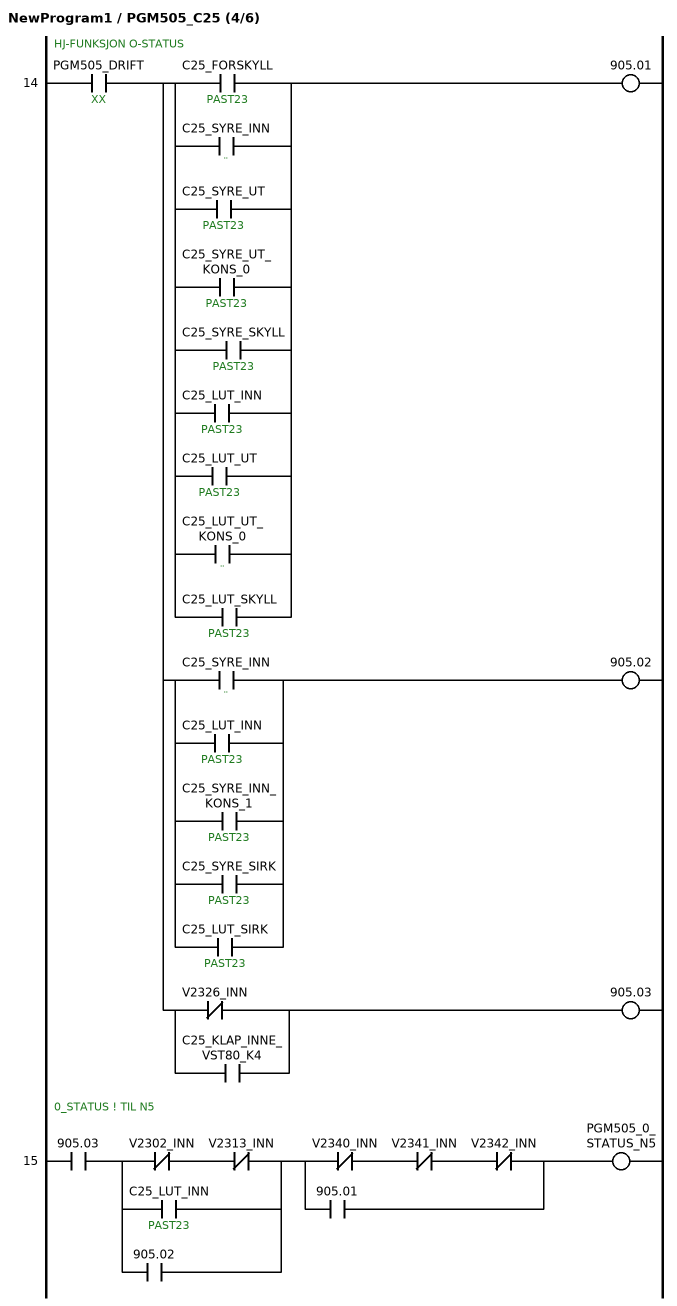
; rung 14: HJ-FUNKSJON O-STATUS
LD PGM505_DRIFT  ; XX
OUT TR0
LD C25_FORSKYLL  ; PAST23
OR C25_SYRE_INN  ; ¨
OR C25_SYRE_UT  ; PAST23
OR C25_SYRE_UT_KONS_0  ; PAST23
OR C25_SYRE_SKYLL  ; PAST23
OR C25_LUT_INN  ; PAST23
OR C25_LUT_UT  ; PAST23
OR C25_LUT_UT_KONS_0  ; ¨
OR C25_LUT_SKYLL  ; PAST23
ANDLD
OUT 905.01
LD TR0
LD C25_SYRE_INN  ; ¨
OR C25_LUT_INN  ; PAST23
OR C25_SYRE_INN_KONS_1  ; PAST23
OR C25_SYRE_SIRK  ; PAST23
OR C25_LUT_SIRK  ; PAST23
ANDLD
OUT 905.02
LD TR0
LDNOT V2326_INN
OR C25_KLAP_INNE_VST80_K4
ANDLD
OUT 905.03
; rung 15: 0_STATUS ! TIL N5
LD 905.03
LDNOT V2302_INN
ANDNOT V2313_INN
OR C25_LUT_INN  ; PAST23
OR 905.02
ANDLD
LDNOT V2340_INN
ANDNOT V2341_INN
ANDNOT V2342_INN
OR 905.01
ANDLD
OUT PGM505_0_STATUS_N5

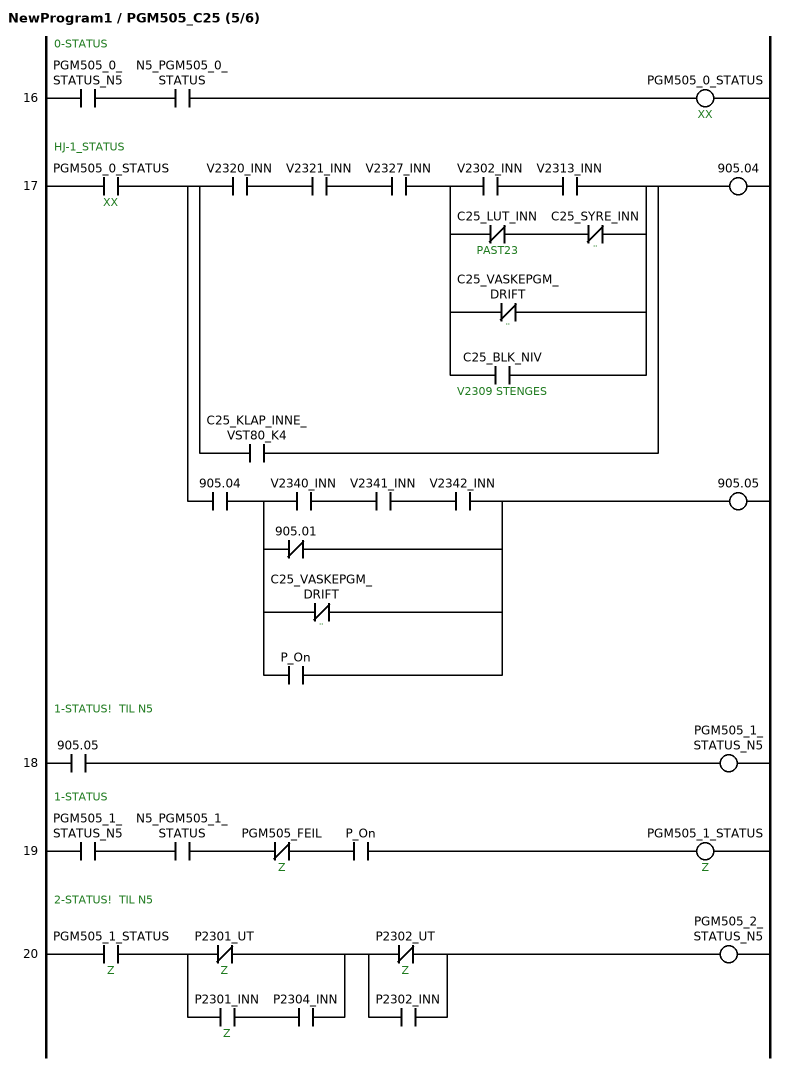
; rung 16: 0-STATUS
LD PGM505_0_STATUS_N5
AND N5_PGM505_0_STATUS
OUT PGM505_0_STATUS  ; XX
; rung 17: HJ-1_STATUS
LD PGM505_0_STATUS  ; XX
OUT TR0
LD V2320_INN
AND V2321_INN
AND V2327_INN
LD V2302_INN
AND V2313_INN
LDNOT C25_LUT_INN  ; PAST23
ANDNOT C25_SYRE_INN  ; ¨
ORLD
ORNOT C25_VASKEPGM_DRIFT  ; ¨
OR C25_BLK_NIV  ; V2309 STENGES
ANDLD
OR C25_KLAP_INNE_VST80_K4
ANDLD
OUT 905.04
LD TR0
AND 905.04
LD V2340_INN
AND V2341_INN
AND V2342_INN
ORNOT 905.01
ORNOT C25_VASKEPGM_DRIFT  ; ¨
OR P_On
ANDLD
OUT 905.05
; rung 18: 1-STATUS!  TIL N5
LD 905.05
OUT PGM505_1_STATUS_N5
; rung 19: 1-STATUS
LD PGM505_1_STATUS_N5
AND N5_PGM505_1_STATUS
ANDNOT PGM505_FEIL  ; Z
AND P_On
OUT PGM505_1_STATUS  ; Z
; rung 20: 2-STATUS!  TIL N5
LD PGM505_1_STATUS  ; Z
LDNOT P2301_UT  ; Z
LD P2301_INN  ; Z
AND P2304_INN
ORLD
ANDLD
LDNOT P2302_UT  ; Z
OR P2302_INN
ANDLD
OUT PGM505_2_STATUS_N5

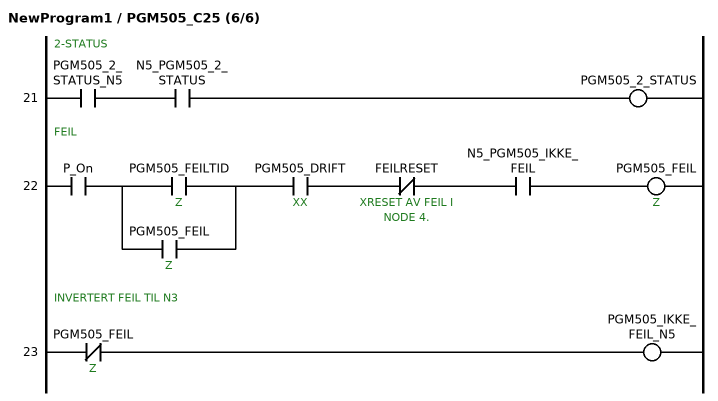
; rung 21: 2-STATUS
LD PGM505_2_STATUS_N5
AND N5_PGM505_2_STATUS
OUT PGM505_2_STATUS
; rung 22: FEIL
LD P_On
LD PGM505_FEILTID  ; Z
OR PGM505_FEIL  ; Z
ANDLD
AND PGM505_DRIFT  ; XX
ANDNOT FEILRESET  ; XRESET AV FEIL I NODE 4.
AND N5_PGM505_IKKE_FEIL
OUT PGM505_FEIL  ; Z
; rung 23: INVERTERT FEIL TIL N3
LDNOT PGM505_FEIL  ; Z
OUT PGM505_IKKE_FEIL_N5
; rung 24: Ingen_kommentar_funnet

### Section C25_KLAPRING

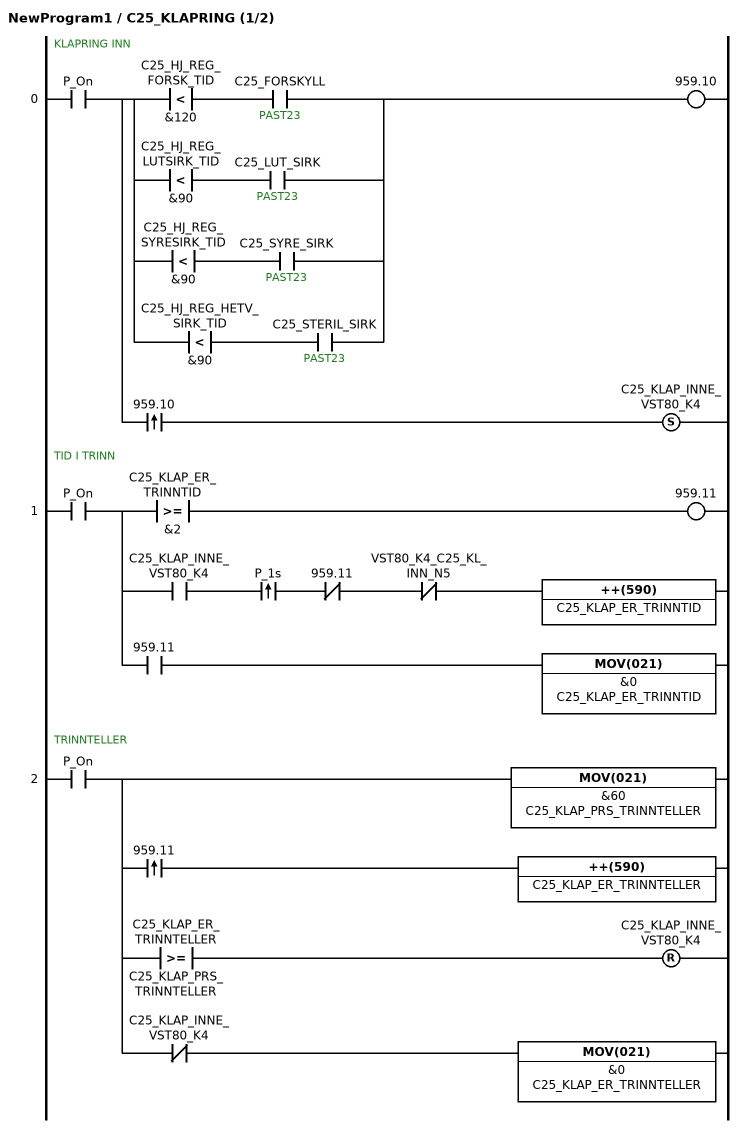
; rung 0: KLAPRING INN
LD P_On
OUT TR0
LD<(310) C25_HJ_REG_FORSK_TID &120
AND C25_FORSKYLL  ; PAST23
LD<(310) C25_HJ_REG_LUTSIRK_TID &90
AND C25_LUT_SIRK  ; PAST23
ORLD
LD<(310) C25_HJ_REG_SYRESIRK_TID &90
AND C25_SYRE_SIRK  ; PAST23
ORLD
LD<(310) C25_HJ_REG_HETV_SIRK_TID &90
AND C25_STERIL_SIRK  ; PAST23
ORLD
ANDLD
OUT 959.10
LD TR0
@AND 959.10
SET C25_KLAP_INNE_VST80_K4
; rung 1: TID I TRINN
LD P_On
OUT TR0
AND>=(325) C25_KLAP_ER_TRINNTID &2
OUT 959.11
LD TR0
AND C25_KLAP_INNE_VST80_K4
@AND P_1s
ANDNOT 959.11
ANDNOT VST80_K4_C25_KL_INN_N5
++(590) C25_KLAP_ER_TRINNTID
LD TR0
AND 959.11
MOV(021) &0 C25_KLAP_ER_TRINNTID
; rung 2: TRINNTELLER
LD P_On
OUT TR0
MOV(021) &60 C25_KLAP_PRS_TRINNTELLER
@AND 959.11
++(590) C25_KLAP_ER_TRINNTELLER
LD TR0
AND>=(325) C25_KLAP_ER_TRINNTELLER C25_KLAP_PRS_TRINNTELLER
RSET C25_KLAP_INNE_VST80_K4
LD TR0
ANDNOT C25_KLAP_INNE_VST80_K4
MOV(021) &0 C25_KLAP_ER_TRINNTELLER

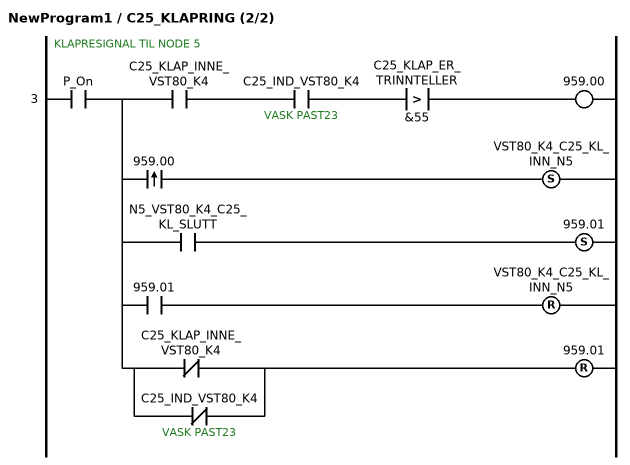
; rung 3: KLAPRESIGNAL TIL NODE 5
LD P_On
OUT TR0
AND C25_KLAP_INNE_VST80_K4
AND C25_IND_VST80_K4  ; VASK PAST23
AND>(320) C25_KLAP_ER_TRINNTELLER &55
OUT 959.00
LD TR0
@AND 959.00
SET VST80_K4_C25_KL_INN_N5
LD TR0
AND N5_VST80_K4_C25_KL_SLUTT
SET 959.01
LD TR0
AND 959.01
RSET VST80_K4_C25_KL_INN_N5
LD TR0
LDNOT C25_KLAP_INNE_VST80_K4
ORNOT C25_IND_VST80_K4  ; VASK PAST23
ANDLD
RSET 959.01
; rung 4: Ingen_kommentar_funnet

### Section PGM_520_BIL01_L1_1_TIL_SILO

